// TwinCAT 3 PLC project WP_Controller
// ProgramVersion: 3.1.4024.0
// libraries:
//   Tc2_MC2, * (Beckhoff Automation GmbH)
//   Tc2_ModbusRTU, * (Beckhoff Automation GmbH)
//   Tc2_Standard, * (Beckhoff Automation GmbH)
//   Tc2_System, * (Beckhoff Automation GmbH)
//   Tc2_Utilities, * (Beckhoff Automation GmbH)
//   Tc3_Module, * (Beckhoff Automation GmbH)
//   Tc3_Vision, * (Beckhoff Automation GmbH)
// project tree:
//   GVLs/ GVL.TcGVL
//   / PlcTask.TcTTO, VisionTask.TcTTO
//   POUs/ FB_ClockPulse.TcPOU (not stored), FB_EnableAxes.TcPOU, FB_StrASCConversion.TcPOU, F_Scale.TcPOU (not stored), MAIN.TcPOU, PRG_LoadcellScaling.TcPOU (not stored), PRG_PLCModbusRTU.TcPOU, PRG_MotorDrive.TcPOU, PRG_PneumaticValves.TcPOU (not stored), PRG_PowerMeasurement.TcPOU, PRG_SafetyLightCurtain.TcPOU, PRG_Thermocouple.TcPOU, PRG_VfdModbusRtu.TcPOU, VISION.TcPOU
// real-time tasks:
//   TASK PlcTask: cycle T#10ms, priority 20, ADS port 350
//   TASK VisionTask: cycle T#10ms, priority 21, ADS port 351
//   TASK VnTask ImgAcq (FileSource1): cycle T#10ms, priority 5, ADS port 352
// motion (NC):
//   TASK NC-Task 1 SAF: cycle T#2ms, priority 4, ADS port 501
//   TASK NC-Task 1 SVB: cycle T#10ms, priority 8, ADS port 511
//   AXIS Axis 1 (id 1)
//     OtherSettings: AllowMotionCmdToSlave=true
//     encoder EncType=1
//     drive DrvType=5
//       Analog: TorqueSetpointScale=10, ScaleFactorActTorque=0.1
//       TimeComp: TaskDelayCycles=1
//     controller CtrType=1
//       CtrPara: PriorControlFactor=1
//         Observer: BandWidth=20
// I/O:
//   DEVICE Device 1 (EtherCAT), AmsNetId 5.57.207.132.2.1
//     Term 1 (EK1200) [EK1200-5000 EtherCAT Power supply (2A E-Bus)]
//       Term 2 (EL1014) [EL1014 4Ch. Dig. Input 24V, 10µs]
//       Term 3 (EL2014) [EL2014 4Ch. Dig. Output 24V, 0,5A, Diagnostic]
//       Term 4 (EL6910) [EL6910, TwinSAFE PLC]
//       Term 5 (EL1904) [EL1904, 4 Ch. Safety Input 24V, TwinSAFE]
//         modules: Module 1 (FSOES)
//       Term 6 (EL3102) [EL3102 2Ch. Ana. Input +/-10V, Diff.]
//       Term 7 (EL4102) [EL4102 2Ch. Ana. Output  0-10V, 16bit]
//       Term 8 (EL9512) [EL9512 Power supply terminal 12V]
//       Term 9 (EL3356-0010) [EL3356-0010 1Ch. Ana. Input Resistor Bridge Terminal, 24bit, High Precision]
//       Term 10 (EL6021) [EL6021 Interface (RS422/485)]
//       Term 11 (EK1110) [EK1110 EtherCAT extension]
//     Term 12 (EK1818) [EK1818 EtherCAT IO-Coupler  (1A E-Bus, 8 Ch. Dig. In, 3ms, 4 Ch. Dig. Out 24V, 0,5A)]
//       Term 13 (EL1809) [EL1809 16Ch. Dig. Input 24V, 3ms]
//       Term 14 (EL2809) [EL2809 16Ch. Dig. Output 24V, 0.5A]
//       Term 15 (EL2904) [EL2904, 4 Ch. Safety Output 24V, 0.5A, TwinSAFE]
//         modules: Module 1 (FSOES), Module 2 (DO)
//       Term 16 (EL9110) [EL9110 Power Supplier with LED (24V, Diagnostics)]
//       Term 17 (EL7031) [EL7031 1Ch. Stepper motor output stage (24V, 1.5A)]
//       Term 18 (EL7201-9014) [EL7201-9014 1Ch. MDP742 Servo motor output stage with OCT (50V, 2.8A RMS) and STO input]
//       Term 19 (EL9011) [EL9011 End Terminal]
// variable links:
//   Device 1 (EtherCAT) <-> Device 1 (EtherCAT)/Term 1 (EK1200)/Term 4 (EL6910)
//     Term 12 (EK1818)/Term 15 (EL2904)/Module 1 (FSOES)/RxPDO/FSOE <-> ConnectionInputs/Message_10 TxPDO
//   Device 1 (EtherCAT) <-> Device 1 (EtherCAT)/Term 1 (EK1200)/Term 5 (EL1904)
//     Term 1 (EK1200)/Term 4 (EL6910)/ConnectionInputs/Message_3 TxPDO <-> Module 1 (FSOES)/RxPDO/FSOE
//     Term 1 (EK1200)/Term 4 (EL6910)/ConnectionOutputs/Message_3 RxPDO <-> Module 1 (FSOES)/TxPDO/FSOE
//   Device 1 (EtherCAT) <-> Device 1 (EtherCAT)/Term 12 (EK1818)/Term 15 (EL2904)
//     Term 1 (EK1200)/Term 4 (EL6910)/ConnectionOutputs/Message_10 RxPDO <-> Module 1 (FSOES)/TxPDO/FSOE
//   WP_Controller/WP_Controller Instance <-> Device 1 (EtherCAT)/Term 1 (EK1200)/Term 4 (EL6910)
//     VisionTask Inputs/GVL.bSafeCommErr <-> StandardInputs/Standard Out Var 7
//     VisionTask Inputs/GVL.bSafeFBErr <-> StandardInputs/Standard Out Var 6
//     VisionTask Inputs/GVL.bSafeRedLedInput <-> StandardInputs/Standard Out Var 8
//     VisionTask Outputs/GVL.bSafeAck <-> StandardOutputs/Standard In Var 1
//     VisionTask Outputs/GVL.bSafeRun <-> StandardOutputs/Standard In Var 2
//   WP_Controller/WP_Controller Instance <-> NC-Task 1 SAF/Axes/Axis 1
//     PlcTask Inputs/GVL.stAxis1.NcToPlc <-> Outputs/ToPlc
//     PlcTask Outputs/GVL.stAxis1.PlcToNc <-> Inputs/FromPlc

CONFIGURATION WP_Controller
    RESOURCE PLC ON TwinCAT3
        TASK PlcTask(INTERVAL := T#10ms, PRIORITY := 20);
        TASK VisionTask(INTERVAL := T#10ms, PRIORITY := 21);
        PROGRAM MAIN WITH PlcTask : MAIN;
        PROGRAM VISION WITH VisionTask : VISION;
    END_RESOURCE
END_CONFIGURATION

// ---- GVLs/GVL.TcGVL
{attribute 'qualified_only'}
VAR_GLOBAL
	//Thermocouple
	nTemp AT %I*: INT;
	
	//Power measurement
	// RMS Current
	fIL1 AT %I*: REAL;
	fIL2 AT %I*: REAL;
	fIL3 AT %I*: REAL;
	
	//RMS Voltage
	fUL1 AT %I*: REAL;
	fUL2 AT %I*: REAL;
	fUL3 AT %I*: REAL;
	
	//Active Power
	fActivePower AT %I* : REAL;
	
	// Phase angle
	fcosphi1 AT %I*: REAL;
	fcosphi2 AT %I*: REAL;
	fcosphi3 AT %I*: REAL;
	
	// Frequency
	fFrequency AT %I*: REAL;
	
	//Motor drive
	stAxis1: AXIS_REF;
	bButtonFw AT %I*: BOOL; //Self reset
	bButtonBw AT %I*: BOOL; //Self reset
	bButtonHalt AT %I*: BOOL; //Self reset
	bButtonAuto AT %I*: BOOL; //Latch
	
	//VFD Modbus RTU
	bEnable AT %I*: BOOL; //Self reset
	bDisable AT %I*: BOOL; //Self reset
	
	// Bit 0 and Bit 1 declaration
	bModbusCoilBit0 : BOOL;
	bModbusCoilBit1 : BOOL;
	
	// Virtual toggle buttons for write values using MODBUS RTU
	bExecuteWriteCoils: BOOL:=TRUE;
	bExecuteWriteRegs0: BOOL;
	//bExecuteWriteRegs1: BOOL;

	// Input STRING from HMI, MAXIMUM 20 characters
	sInputFromHMI: STRING(20);		

	//Constant value for testing, used for EL2596
	bLedEnable AT %Q*:BOOL:=TRUE;
	bLedOutput AT %Q*:BOOL:=TRUE;
	bOutputCurrent AT %Q*: UINT:=300;
	
	// Constant value for EL2809 controlling strobe
	bLedEnableEL2xxx AT %Q*:BOOL:=TRUE; 
	
	// Loadcell scaling variables
	uLoadCellRawValue AT %I*: DINT;
	uLoadCellScaledValue: REAL;
	
	// Output signal variables for sneumatic valves 
	bValve1 AT %Q*:BOOL;
	bValve2 AT %Q*:BOOL;
	bValve3 AT %Q*:BOOL;
	bValve4 AT %Q*:BOOL;
	bValve5 AT %Q*:BOOL;
	bValve6 AT %Q*:BOOL;
	bVirtualToggleButton1:BOOL;
	bVirtualToggleButton2:BOOL;
	bVirtualToggleButton3:BOOL;
	bVirtualToggleButton4:BOOL;
	bVirtualToggleButton5:BOOL;
	bVirtualToggleButton6:BOOL;
	
	// TwinSAFE declaration
	bSafeRun AT %Q*:BOOL;
	bSafeAck AT %Q*:BOOL;
	bSafeFBErr AT %I*: BOOL;
	bSafeCommErr AT %I*: BOOL;
	bSafeRedLedOutput AT %Q*:BOOL; // safety output signal for EL2809 
	bSafeRedLedInput AT %I*:BOOL; // safety red led reception signal for ouput signal imported from EL6910	
	
	
END_VAR

// ---- POUs/MAIN.TcPOU
PROGRAM MAIN
VAR
END_VAR

PRG_Thermocouple();
PRG_PowerMeasurement();
PRG_MotorDrive();
PRG_PneumaticValves();
PRG_PLCModbusRTU();
PRG_LoadcellScaling();

END_PROGRAM

// ---- POUs/PRG_Thermocouple.TcPOU
PROGRAM PRG_Thermocouple
VAR
	fTemp: REAL;
END_VAR

fTemp := GVL.nTemp;

END_PROGRAM

// ---- POUs/PRG_PowerMeasurement.TcPOU
PROGRAM PRG_PowerMeasurement
VAR
	fActivePowerAbs: REAL;
	fIL1Abs: REAL;
	fIL2Abs: REAL;
	fIL3Abs: REAL;
END_VAR

fActivePowerAbs := ABS(GVL.fActivePower);
fIL1Abs := ABS(GVL.fIL1);
fIL2Abs := ABS(GVL.fIL2);
fIL3Abs := ABS(GVL.fIL3);

END_PROGRAM

// ---- POUs/PRG_MotorDrive.TcPOU
PROGRAM PRG_MotorDrive
VAR
	fbEnableAxes: FB_EnableAxes;
	fbHalt1: MC_Halt;
	fbMoveVelocityFw: MC_MoveVelocity;
	fbMoveVelocityBw: MC_MoveVelocity;
	fbTON1: TON;
	fbRTrigMoveFw: R_TRIG;
	fbRTrigMoveBw: R_TRIG;
	fbRTrigHalt: R_TRIG;
	nAutoState: INT;
END_VAR

fbEnableAxes.bEnableAxes := TRUE;
fbRTrigMoveFW(CLK:=GVL.bButtonFw, Q=>);
fbRTrigMoveBW(CLK:=GVL.bButtonBw, Q=>);
fbRTrigHalt(CLK:=GVL.bButtonHalt, Q=>);

IF fbRTrigMoveFw.Q THEN
	fbHalt1.Execute := FALSE;
	fbMoveVelocityBw.Execute := FALSE;
	fbMoveVelocityFw.Execute := TRUE;
END_IF

IF fbRTrigMoveBw.Q THEN
	fbHalt1.Execute := FALSE;
	fbMoveVelocityFw.Execute := FALSE;
	fbMoveVelocityBw.Execute := TRUE;
END_IF

IF fbRTrigHalt.Q THEN
	fbHalt1.Execute := TRUE;
	fbMoveVelocityFw.Execute := FALSE;
	fbMoveVelocityBw.Execute := FALSE;
END_IF

IF GVL.bButtonAuto THEN
	CASE nAutoState OF
		0: //Initialize auto motion
			fbHalt1.Execute := FALSE;
			fbMoveVelocityFw.Execute := FALSE;
			fbMoveVelocityBw.Execute := FALSE;
			nAutoState := 1;
		1: //Move forward
			fbTON1(IN:=TRUE, PT:=T#4S, Q=>, ET=>);
			fbMoveVelocityFw.Execute := TRUE;
			IF fbTON1.Q THEN
				fbTON1(IN:=FALSE);
				nAutoState := 2;	
			END_IF
		2: //Halt
			fbTON1(IN:=TRUE, PT:=T#2S, Q=>, ET=>);
			fbMoveVelocityFw.Execute := FALSE;
			fbHalt1.Execute := TRUE;
			IF fbTON1.Q THEN
				fbTON1(IN:=FALSE);
				nAutoState := 3;	
			END_IF
		3: //Move backward
			fbTON1(IN:=TRUE, PT:=T#4S, Q=>, ET=>);
			fbHalt1.Execute := FALSE;
			fbMoveVelocityBw.Execute := TRUE;
			IF fbTON1.Q THEN
				fbTON1(IN:=FALSE);
				nAutoState := 4;	
			END_IF
		4: //Halt again
			fbTON1(IN:=TRUE, PT:=T#2S, Q=>, ET=>);
			fbMoveVelocityBw.Execute := FALSE;
			fbHalt1.Execute := TRUE;
			IF fbTON1.Q THEN
				fbTON1(IN:=FALSE);
				nAutoState := 0;	
			END_IF
	END_CASE
END_IF

A_EnableAxes();
A_MoveVelocityFw();
A_MoveVelocityBw();
A_Halt();

ACTION A_EnableAxes:
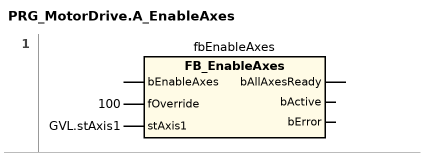
// NETWORK 1
fbEnableAxes(fOverride := 100, stAxis1 := GVL.stAxis1); // FB_EnableAxes
END_ACTION

ACTION A_Halt:
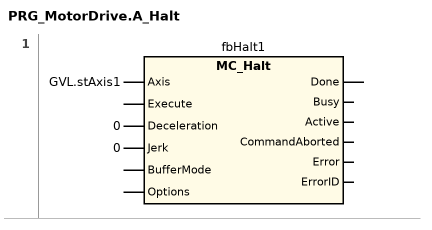
// NETWORK 1
fbHalt1(Axis := GVL.stAxis1, Deceleration := 0, Jerk := 0); // MC_Halt
END_ACTION

ACTION A_MoveVelocityBw:
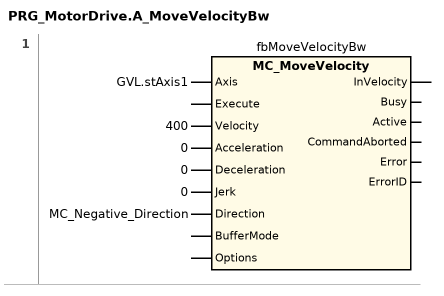
// NETWORK 1
fbMoveVelocityBw(
    Axis := GVL.stAxis1,
    Velocity := 400,
    Acceleration := 0,
    Deceleration := 0,
    Jerk := 0,
    Direction := MC_Negative_Direction); // MC_MoveVelocity
END_ACTION

ACTION A_MoveVelocityFw:
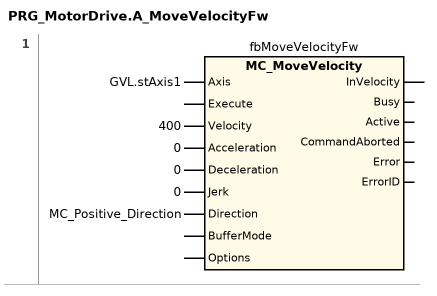
// NETWORK 1
fbMoveVelocityFw(
    Axis := GVL.stAxis1,
    Velocity := 400,
    Acceleration := 0,
    Deceleration := 0,
    Jerk := 0,
    Direction := MC_Positive_Direction); // MC_MoveVelocity
END_ACTION

END_PROGRAM

// ---- POUs/FB_EnableAxes.TcPOU
FUNCTION_BLOCK FB_EnableAxes
VAR_INPUT
	bEnableAxes			: BOOL;
	fOverride			: LREAL;
END_VAR
VAR_OUTPUT
	bAllAxesReady		: BOOL;
	bActive				: BOOL;
	bError				: BOOL;
END_VAR
VAR_IN_OUT
	stAxis1				: AXIS_REF;
END_VAR
VAR
	fbPower1			:MC_Power;
END_VAR

fbPower1(
	Enable:=bEnableAxes, 
	Enable_Positive:=bEnableAxes, 
	Enable_Negative:=bEnableAxes, 
	Override:=fOverride, 
	BufferMode:= , 
	Axis:=stAxis1, 
	Status=> , 
	Busy=> , 
	Active=> , 
	Error=> , 
	ErrorID=> );

IF fbPower1.Active THEN
	bActive := TRUE;
	IF fbPower1.Error THEN
		bError := TRUE;
	ELSE 
		bAllAxesReady := fbPower1.Status;
		bError := FALSE;
	END_IF
ELSE
	bActive := FALSE;
END_IF

END_FUNCTION_BLOCK

// ---- POUs/PRG_PLCModbusRTU.TcPOU
PROGRAM PRG_PLCModbusRTU
VAR
	fbStrAscConversion: FB_StrASCConversion;
	fbClockPulse: FB_ClockPulse; // 200ms pulse
	fbModbusMaster: ModbusRtuMasterV2_KL6x22B;
	sWriteErrorId: MODBUS_ERRORS;
	bBusyState: BOOL := FALSE;

	// Modbus properties
	mB_quantity_coils: WORD:=2;
	mB_quantity_regs: WORD:=20;
	mB_addr_bits: WORD:=00;
	mB_addr_regs: WORD:=40;

	
	// Holding register declaration
	aWriteValueRegs0: ARRAY[0..19] OF WORD;
	
	// Compressed form of coil registers
	wWriteValueBits: WORD; //BIT0|BIT1|XXXXXXXXX

	bExecuteClockPulse: BOOL;
END_VAR

fbClockPulse(bStart:= GVL.bExecuteWriteCoils, bExecute => bExecuteClockPulse);

// Convert STRING to ARRAY OF BYTE in ASCII TYPE
fbStrAscConversion(sText:=GVL.sInputFromHMI,aASCIIRes => aWriteValueRegs0);

// Convert Bit 0 and Bit 1 to WORD
wWriteValueBits := M_BoolWordConversion();

A_WriteCoils();
A_WriteRegs();

ACTION A_WriteCoils:
// Write coils
	fbModbusMaster.WriteMultipleCoils(
	UnitID:= 10, 
	Quantity:= mB_quantity_coils, 
	MBAddr:= mB_addr_bits, 
	cbLength:= SIZEOF(wWriteValueBits), 
	pMemoryAddr:= ADR(wWriteValueBits), 
	Execute:= bExecuteClockPulse, 
	Timeout:= T#2S, 
	BUSY=> bBusyState, 
	Error=> , 
	ErrorId=> sWriteErrorId, 
	cbRead=>
	);
END_ACTION

ACTION A_WriteRegs:

// Write 1st register
	fbModbusMaster.WriteRegs(
	UnitID:= 10, 
	Quantity:= mB_quantity_regs, 
	MBAddr:= mB_addr_regs, 
	cbLength:= SIZEOF(aWriteValueRegs0), 
	pMemoryAddr:= ADR(aWriteValueRegs0), 
	Execute:= GVL.bExecuteWriteRegs0, 
	Timeout:= T#2S, 
	BUSY=> bBusyState, 
	Error=> , 
	ErrorId=> sWriteErrorId, 
	cbRead=>
	);
END_ACTION

METHOD M_BoolWordConversion : WORD
VAR_INPUT
END_VAR
IF GVL.bModbusCoilBit0 THEN
	IF GVL.bModbusCoilBit1 THEN
		M_BoolWordConversion := 3;
	ELSE
		M_BoolWordConversion := 1;
	END_IF
ELSE
	IF GVL.bModbusCoilBit1 THEN
		M_BoolWordConversion := 2;
	ELSE
		M_BoolWordConversion := 0;
	END_IF
END_IF
END_METHOD

END_PROGRAM

// ---- POUs/FB_StrASCConversion.TcPOU
FUNCTION_BLOCK FB_StrASCConversion
VAR_INPUT
	sText : STRING(20):='00000000000000000000';
END_VAR
VAR_OUTPUT
	aASCIIRes : ARRAY[0..19] OF WORD;
END_VAR
VAR
	words: ARRAY[0..19] OF BYTE;
	currentString:STRING(1):='';
	nCount:INT:=0;
	nCountConvert: INT:=0;
END_VAR

FOR nCount := 0 TO 20 BY 1 DO
	currentString[0]:=sText[nCount];
	words[nCount]:=currentString[0] ;
	aASCIIRes[nCount]:=words[nCount];
END_FOR

END_FUNCTION_BLOCK

// ---- POUs/VISION.TcPOU
PROGRAM VISION
VAR
	hr					: HRESULT;
	
	fbControl			: FB_VN_GevCameraControl;
	eState				: ETcVnCameraState;
	
	// Image
	ipImage				: ITcVnImage;
	ipImageWork			: ITcVnImage;
	ipImageResult		: ITcVnImage;
	
	// displayable Image
	ipImageDispl		: ITcVnDisplayableImage;
	ipImageWorkDispl	: ITcVnDisplayableImage;
	ipImageResultDispl	: ITcVnDisplayableImage;
	
	// QR Code
	ipCodeDecodedList   :    ITcVnContainer; 
	ipCodeContourList   :    ITcVnContainer;
	sCodeAsString       :    STRING(255);
	sErrorString		:	 STRING(255);
	eBarcodeSearchDirection   :   ETcVnBarcodeSearchDirection := TCVN_BSD_ANY;
	eBarcodeType              :   ETcVnBarcodeType := TCVN_BT_EAN13;


	// Watchdog
	hrWD                :    HRESULT;
	//tStop               :    DINT := 20000; //qr code
	tStop               :    DINT := 50000; //qr code
	tRest               :    DINT;

	// Color
	aRedColor           :    TcVnVector4_LREAL := [255, 0, 0];
	aGreenColor			:	 TcVnVector4_LREAL := [0, 255, 0];

	// Return code
	nReturnCode               :   DWORD;
	sReturnCode               :   STRING;
	sResultText               :   STRING;
END_VAR

eState := fbControl.GetState();

CASE eState OF
	TCVN_CS_INITIAL, 			(* The camera controller is in the initial state and ready to establish the connection to the camera. *)
	TCVN_CS_INITIALIZING, 		(* The camera controller is initializing the camera. *)
	TCVN_CS_INITIALIZED, 		(* The camera controller has initialized the camera. *)
	TCVN_CS_OPENING, 			(* The camera controller is establishing the connection to the camera. *)
	TCVN_CS_OPENED, 			(* The connection to the camera has been established and the camera controller is ready to start the image acquisition. *)
	TCVN_CS_STARTACQUISITION: 	(* The camera controller is starting the image acquisition. *)
	
		hr := fbControl.StartAcquisition();
	
	TCVN_CS_ACQUIRING: 			(* The camera is sending images (either streaming or manually triggered, depending on the configuration). *)
	
		hr := fbControl.GetCurrentImage(ipImage);
		IF  SUCCEEDED(hr) THEN
			sCodeAsString :='Scanning... No code found!';
			// Conver color space from grayscale to RGB, Display input image (without processing)
			hr:=F_VN_ConvertColorSpace(ipImage,ipImageResult,ETcVnColorSpaceTransform.TCVN_CST_GRAY_TO_RGB,hr);
			hr:=F_VN_CopyImage(ipImageResult,ipImageWork,hr);
			hr:= F_VN_CopyIntoDisplayableImage(ipSrcImage:= ipImage,ipDestImage:=ipImageDispl,hrPrev:=hr);
			// Pre result image processing
			hr := F_VN_PutTextExp(sCodeAsString, ipImageWork, 50, 100, TCVN_FT_HERSHEY_PLAIN, 5, aRedColor,3, TCVN_LT_4_CONNECTED, FALSE, hr);
			hr:=F_VN_CopyIntoDisplayableImage(ipSrcImage:= ipImageWork,ipDestImage:=ipImageResultDispl,hrPrev:=hr);

			// Execute the Barcode Reading Function with EAN13 selected monitored by the Watchdog-Function
			hrWD := F_VN_StartRelWatchdog(tStop, hr);
			(*hr := F_VN_ReadQRCodeExp(
            ipSrcImage      :=  ipImage,
            ipDecodedData   :=  ipCodeDecodedList,
            ipContours      :=  ipCodeContourList,
            nCodeNumber     :=  1,
            eSearchStrategy :=  TCVN_CSS_ONLY_NOT_INVERTED + TCVN_CSS_ONLY_NOT_FLIPPED,
            hrPrev          :=  hr
   			 );*)
	    	hr := F_VN_ReadBarcodeExp(
               ipSrcImage         :=   ipImage,
               ipDecodedData      :=   ipCodeDecodedList,
               ipContours         :=   ipCodeContourList,
               eBarcodeType       :=   eBarcodeType,
               nCodeNumber        :=   1, 
               eSearchDirection   :=   eBarcodeSearchDirection,
               hrPrev             :=   hr);
			hrWD := F_VN_StopWatchdog(hrWD, tRest => tRest);
			//ADSLOGDINT(msgCtrlMask:=ADSLOG_MSGTYPE_MSGBOX,msgFmtStr:='hrResult1 %d',dintArg:=hr);
			// Handle return-code
			IF hr = S_OK THEN
				// Prepare code result in string
				hr := F_VN_ExportSubContainer_String(ipCodeDecodedList, 0, sCodeAsString, 255, hr);
				sCodeAsString := CONCAT('Code: ', sCodeAsString);
			ELSE
				// Check for succeeded return codes or add specific error handling
				CASE hr OF
					S_FALSE: 
						sResultText := 'No code found...'; 
			
					S_WATCHDOG_TIMEOUT: 
						sResultText := 'Cancelled by watchdog...'; 
				ELSE
					// Extract error-code from HRESULT & react accordingly
					nReturnCode := DINT_TO_DWORD(hr) AND 16#FFF; 
					sReturnCode := DWORD_TO_HEXSTR(nReturnCode, 3, FALSE); 
					sResultText := CONCAT('Returncode ', sReturnCode); 
				END_CASE
			END_IF
			
			// Draw Code Contour into Result Image
		    hr := F_VN_DrawContours(ipCodeContourList, 0, ipImageResult, aGreenColor, 3, hr);
			// Write Code into Result Image
    		hr := F_VN_PutTextExp(sCodeAsString, ipImageResult, 50, 100, TCVN_FT_HERSHEY_PLAIN, 5, aGreenColor,3, TCVN_LT_4_CONNECTED, FALSE, hr);
			// Write Code Reading proceeded time into Result Image
			//sText := CONCAT(CONCAT('Time: ', DINT_TO_STRING(tStop - tRest)), 'us');
			hr := F_VN_TransformIntoDisplayableImage(ipSrcImage:=ipImageResult, ipDestImage:=ipImageResultDispl, hrPrev:=hr);
		END_IF
		

	TCVN_CS_ERROR: 	(* The camera controller is in an error state (e.g. the connection to the camera was lost). *)
		fbControl.Reset();
END_CASE

END_PROGRAM

// ---- POUs/PRG_SafetyLightCurtain.TcPOU
PROGRAM PRG_SafetyLightCurtain
VAR
END_VAR

GVL.bSafeRedLedOutput := GVL.bSafeRedLedInput;

END_PROGRAM

// ---- POUs/PRG_VfdModbusRtu.TcPOU
PROGRAM PRG_VfdModbusRtu
VAR
	fbVfdMb: ModbusRtuMaster_KL6x22B;
	fbRTrigWrite: R_Trig;
	fbRTrigEnable: R_Trig;
	fbRTrigDisable: R_Trig;
	fbTON: TON;
	wQty: WORD := 1;
	wMbAddr: WORD;
	wCmd: WORD;
	bWrite: BOOL;
END_VAR

fbRTrigWrite(CLK:=bWrite, Q=>);
fbRTrigEnable(CLK:=GVL.bEnable, Q=>);
fbRTrigEnable(CLK:=GVL.bDisable, Q=>);

IF fbRTrigEnable.Q THEN
	bWrite := TRUE;
	fbTON(IN:= bWrite, PT:= T#500MS, Q=> , ET=> );
	wMbAddr := 416;
	wCmd := 1;
END_IF

IF fbRTrigDisable.Q THEN
	bWrite := TRUE;
	fbTON(IN:= bWrite, PT:= T#500MS, Q=> , ET=> );
	wMbAddr := 416;
	wCmd := 0;
END_IF

IF fbTON.Q THEN
	fbTON(IN:=FALSE);
	bWrite := FALSE;
END_IF

fbVfdMb.WriteRegs(
	UnitID:= 1, 
	Quantity:= wQty, 
	MBAddr:= wMbAddr, 
	cbLength:= SIZEOF(wCmd), 
	pMemoryAddr:= ADR(wCmd), 
	Execute:= fbRTrigWrite.Q, 
	Timeout:= T#1S, 
	BUSY=> , 
	Error=> , 
	ErrorId=> , 
	cbRead=> );

END_PROGRAM
